TYPE ST_Module_CtrlStatus_Base :
STRUCT
	HeartbeatIndex : UDINT;
	ModuleCtrl : ST_ModuleCtrl;
	ModuleStatus : ST_ModuleStatus;
	ModuleVariableList : ARRAY[1..Param_Config.MaxModuleVariable] OF ST_ExtDescriptor;
	ModuleAlarmList : ARRAY[1..Param_Config.MaxPublishedModuleAlarms] OF ST_ExtAlarm;
	ModuleDataList : ARRAY[1..Param_Config.MaxModuleData] OF ST_ExtDescriptor;
END_STRUCT
END_TYPE

(* stored: Version 1.1.0.1, ProductVersion 3.1.4026.18
   DUT ST_Module_CtrlStatus_Base: Id {fb4253f3-2644-4b9d-bb36-cb86132b772d} *)
